// TIA Portal V17 export
// export: Created 2023-08-28T22:41:32.6164324Z, ExportSetting WithDefaults, DisplayName Totally Integrated Automation Portal, DisplayVersion V17 Update 5, DisplayName TIA Portal Openness, DisplayVersion V17 Update 5, DisplayName TIA Portal Teamcenter Gateway, DisplayVersion V17 Update 5, DisplayName TIA Portal Version Control Interface, DisplayVersion V17, DisplayName Simotion SCOUT TIA, DisplayVersion 5.4.3.0, DisplayName TIA Portal Test Suite Advanced, DisplayVersion V17 Update 1, DisplayName SIMOCODE ES, DisplayVersion V17 Update 5, DisplayName SINAMICS Startdrive Advanced, DisplayVersion V17 SP1, DisplayName SINAMICS Startdrive G130, G150, S120, S150, SINAMICS MV, S210, DisplayVersion V17 SP1, DisplayName SINAMICS Startdrive G110M, G120, G120C, G120D, G120P, G115D, DisplayVersion V17 SP1, DisplayName SIRIUS Safety ES, DisplayVersion V17 Update 5, DisplayName STEP 7 Professional, DisplayVersion V17 Update 5, DisplayName STEP 7 CFC, DisplayVersion V17 Update 1, DisplayName STEP 7 Safety, DisplayVersion V17, DisplayName WinCC Advanced, DisplayVersion V17 Update 5, DisplayName SIMATIC Visualization Architect, DisplayVersion V17 Update 5
DATA_BLOCK "S1.CABINET000.STATE"   // DB2700
// stored: AutoNumber true, DBAccessibleFromOPCUA true, DBAccessibleFromWebserver true, InstanceOfName CabState, InstanceOfType FB
"CabState "
BEGIN
END_DATA_BLOCK

DATA_BLOCK "S1.CABINET001.STATE"   // DB2701
// stored: AutoNumber true, DBAccessibleFromOPCUA true, DBAccessibleFromWebserver true, InstanceOfName CabState, InstanceOfType FB
"CabState "
BEGIN
END_DATA_BLOCK

DATA_BLOCK "S1.CABINET002.STATE"   // DB2702
// stored: AutoNumber true, DBAccessibleFromOPCUA true, DBAccessibleFromWebserver true, InstanceOfName CabState, InstanceOfType FB
"CabState "
BEGIN
END_DATA_BLOCK

DATA_BLOCK "S1.CABINET003.STATE"   // DB2703
// stored: AutoNumber true, DBAccessibleFromOPCUA true, DBAccessibleFromWebserver true, InstanceOfName CabState, InstanceOfType FB
"CabState "
BEGIN
END_DATA_BLOCK

DATA_BLOCK "S1.CABINET004.STATE"   // DB2704
// stored: AutoNumber true, DBAccessibleFromOPCUA true, DBAccessibleFromWebserver true, InstanceOfName CabState, InstanceOfType FB
"CabState "
BEGIN
END_DATA_BLOCK

DATA_BLOCK "S1.CABINET005.STATE"   // DB2705
// stored: AutoNumber true, DBAccessibleFromOPCUA true, DBAccessibleFromWebserver true, InstanceOfName CabState, InstanceOfType FB
"CabState "
BEGIN
END_DATA_BLOCK

DATA_BLOCK "S1.CABINET006.STATE"   // DB2706
// stored: AutoNumber true, DBAccessibleFromOPCUA true, DBAccessibleFromWebserver true, InstanceOfName CabState, InstanceOfType FB
"CabState "
BEGIN
END_DATA_BLOCK

DATA_BLOCK "S1.CABINET007.STATE"   // DB2707
// stored: AutoNumber true, DBAccessibleFromOPCUA true, DBAccessibleFromWebserver true, InstanceOfName CabState, InstanceOfType FB
"CabState "
BEGIN
END_DATA_BLOCK

DATA_BLOCK "S1.CABINET008.STATE"   // DB2708
// stored: AutoNumber true, DBAccessibleFromOPCUA true, DBAccessibleFromWebserver true, InstanceOfName CabState, InstanceOfType FB
"CabState "
BEGIN
END_DATA_BLOCK

DATA_BLOCK "S1.CABINET009.STATE"   // DB2709
// stored: AutoNumber true, DBAccessibleFromOPCUA true, DBAccessibleFromWebserver true, InstanceOfName CabState, InstanceOfType FB
"CabState "
BEGIN
END_DATA_BLOCK

DATA_BLOCK "S1.CABINET010.STATE"   // DB2710
// stored: AutoNumber true, DBAccessibleFromOPCUA true, DBAccessibleFromWebserver true, InstanceOfName CabState, InstanceOfType FB
"CabState "
BEGIN
END_DATA_BLOCK

DATA_BLOCK "S1.CABINET011.STATE"   // DB2711
// stored: AutoNumber true, DBAccessibleFromOPCUA true, DBAccessibleFromWebserver true, InstanceOfName CabState, InstanceOfType FB
"CabState "
BEGIN
END_DATA_BLOCK

DATA_BLOCK "S1.CABINET012.STATE"   // DB2712
// stored: AutoNumber true, DBAccessibleFromOPCUA true, DBAccessibleFromWebserver true, InstanceOfName CabState, InstanceOfType FB
"CabState "
BEGIN
END_DATA_BLOCK

DATA_BLOCK "S1.CABINET013.STATE"   // DB2713
// stored: AutoNumber true, DBAccessibleFromOPCUA true, DBAccessibleFromWebserver true, InstanceOfName CabState, InstanceOfType FB
"CabState "
BEGIN
END_DATA_BLOCK

DATA_BLOCK "S1.CABINET014.STATE"   // DB2714
// stored: AutoNumber true, DBAccessibleFromOPCUA true, DBAccessibleFromWebserver true, InstanceOfName CabState, InstanceOfType FB
"CabState "
BEGIN
END_DATA_BLOCK

DATA_BLOCK "S1.CABINET015.STATE"   // DB2715
// stored: AutoNumber true, DBAccessibleFromOPCUA true, DBAccessibleFromWebserver true, InstanceOfName CabState, InstanceOfType FB
"CabState "
BEGIN
END_DATA_BLOCK

DATA_BLOCK "S1.CABINET016.STATE"   // DB2716
// stored: AutoNumber true, DBAccessibleFromOPCUA true, DBAccessibleFromWebserver true, InstanceOfName CabState, InstanceOfType FB
"CabState "
BEGIN
END_DATA_BLOCK

DATA_BLOCK "S1.CABINET017.STATE"   // DB2717
// stored: AutoNumber true, DBAccessibleFromOPCUA true, DBAccessibleFromWebserver true, InstanceOfName CabState, InstanceOfType FB
"CabState "
BEGIN
END_DATA_BLOCK

DATA_BLOCK "S1.CABINET018.STATE"   // DB2718
// stored: AutoNumber true, DBAccessibleFromOPCUA true, DBAccessibleFromWebserver true, InstanceOfName CabState, InstanceOfType FB
"CabState "
BEGIN
END_DATA_BLOCK

DATA_BLOCK "S1.CABINET019.STATE"   // DB2719
// stored: AutoNumber true, DBAccessibleFromOPCUA true, DBAccessibleFromWebserver true, InstanceOfName CabState, InstanceOfType FB
"CabState "
BEGIN
END_DATA_BLOCK

DATA_BLOCK "S1.CABINET020.STATE"   // DB2720
// stored: AutoNumber true, DBAccessibleFromOPCUA true, DBAccessibleFromWebserver true, InstanceOfName CabState, InstanceOfType FB
"CabState "
BEGIN
END_DATA_BLOCK

DATA_BLOCK "S1.CABINET021.STATE"   // DB2721
// stored: AutoNumber true, DBAccessibleFromOPCUA true, DBAccessibleFromWebserver true, InstanceOfName CabState, InstanceOfType FB
"CabState "
BEGIN
END_DATA_BLOCK

DATA_BLOCK "S1.CABINET022.STATE"   // DB2722
// stored: AutoNumber true, DBAccessibleFromOPCUA true, DBAccessibleFromWebserver true, InstanceOfName CabState, InstanceOfType FB
"CabState "
BEGIN
END_DATA_BLOCK

DATA_BLOCK "S1.CABINET023.STATE"   // DB2723
// stored: AutoNumber true, DBAccessibleFromOPCUA true, DBAccessibleFromWebserver true, InstanceOfName CabState, InstanceOfType FB
"CabState "
BEGIN
END_DATA_BLOCK

DATA_BLOCK "S1.CABINET024.STATE"   // DB2724
// stored: AutoNumber true, DBAccessibleFromOPCUA true, DBAccessibleFromWebserver true, InstanceOfName CabState, InstanceOfType FB
"CabState "
BEGIN
END_DATA_BLOCK

DATA_BLOCK "S1.CABINET025.STATE"   // DB2725
// stored: AutoNumber true, DBAccessibleFromOPCUA true, DBAccessibleFromWebserver true, InstanceOfName CabState, InstanceOfType FB
"CabState "
BEGIN
END_DATA_BLOCK

DATA_BLOCK "S1.CABINET026.STATE"   // DB2726
// stored: AutoNumber true, DBAccessibleFromOPCUA true, DBAccessibleFromWebserver true, InstanceOfName CabState, InstanceOfType FB
"CabState "
BEGIN
END_DATA_BLOCK

DATA_BLOCK "S1.CABINET027.STATE"   // DB2727
// stored: AutoNumber true, DBAccessibleFromOPCUA true, DBAccessibleFromWebserver true, InstanceOfName CabState, InstanceOfType FB
"CabState "
BEGIN
END_DATA_BLOCK

DATA_BLOCK "S1.CABINET028.STATE"   // DB2728
// stored: AutoNumber true, DBAccessibleFromOPCUA true, DBAccessibleFromWebserver true, InstanceOfName CabState, InstanceOfType FB
"CabState "
BEGIN
END_DATA_BLOCK

DATA_BLOCK "S1.CABINET029.STATE"   // DB2729
// stored: AutoNumber true, DBAccessibleFromOPCUA true, DBAccessibleFromWebserver true, InstanceOfName CabState, InstanceOfType FB
"CabState "
BEGIN
END_DATA_BLOCK

DATA_BLOCK "S1.CABINET030.STATE"   // DB2730
// stored: AutoNumber true, DBAccessibleFromOPCUA true, DBAccessibleFromWebserver true, InstanceOfName CabState, InstanceOfType FB
"CabState "
BEGIN
END_DATA_BLOCK

DATA_BLOCK "S1.CABINET031.STATE"   // DB2731
// stored: AutoNumber true, DBAccessibleFromOPCUA true, DBAccessibleFromWebserver true, InstanceOfName CabState, InstanceOfType FB
"CabState "
BEGIN
END_DATA_BLOCK

DATA_BLOCK "S1.CABINET032.STATE"   // DB2732
// stored: AutoNumber true, DBAccessibleFromOPCUA true, DBAccessibleFromWebserver true, InstanceOfName CabState, InstanceOfType FB
"CabState "
BEGIN
END_DATA_BLOCK

DATA_BLOCK "S1.CABINET033.STATE"   // DB2733
// stored: AutoNumber true, DBAccessibleFromOPCUA true, DBAccessibleFromWebserver true, InstanceOfName CabState, InstanceOfType FB
"CabState "
BEGIN
END_DATA_BLOCK

DATA_BLOCK "S1.CABINET034.STATE"   // DB2734
// stored: AutoNumber true, DBAccessibleFromOPCUA true, DBAccessibleFromWebserver true, InstanceOfName CabState, InstanceOfType FB
"CabState "
BEGIN
END_DATA_BLOCK

DATA_BLOCK "S1.CABINET035.STATE"   // DB2735
// stored: AutoNumber true, DBAccessibleFromOPCUA true, DBAccessibleFromWebserver true, InstanceOfName CabState, InstanceOfType FB
"CabState "
BEGIN
END_DATA_BLOCK

DATA_BLOCK "S1.CABINET036.STATE"   // DB2736
// stored: AutoNumber true, DBAccessibleFromOPCUA true, DBAccessibleFromWebserver true, InstanceOfName CabState, InstanceOfType FB
"CabState "
BEGIN
END_DATA_BLOCK

DATA_BLOCK "S1.CABINET037.STATE"   // DB2737
// stored: AutoNumber true, DBAccessibleFromOPCUA true, DBAccessibleFromWebserver true, InstanceOfName CabState, InstanceOfType FB
"CabState "
BEGIN
END_DATA_BLOCK

DATA_BLOCK "S1.CABINET038.STATE"   // DB2738
// stored: AutoNumber true, DBAccessibleFromOPCUA true, DBAccessibleFromWebserver true, InstanceOfName CabState, InstanceOfType FB
"CabState "
BEGIN
END_DATA_BLOCK

DATA_BLOCK "S1.CABINET039.STATE"   // DB2739
// stored: AutoNumber true, DBAccessibleFromOPCUA true, DBAccessibleFromWebserver true, InstanceOfName CabState, InstanceOfType FB
"CabState "
BEGIN
END_DATA_BLOCK

DATA_BLOCK "S1.CABINET040.STATE"   // DB2740
// stored: AutoNumber true, DBAccessibleFromOPCUA true, DBAccessibleFromWebserver true, InstanceOfName CabState, InstanceOfType FB
"CabState "
BEGIN
END_DATA_BLOCK

DATA_BLOCK "S1.CABINET041.STATE"   // DB2741
// stored: AutoNumber true, DBAccessibleFromOPCUA true, DBAccessibleFromWebserver true, InstanceOfName CabState, InstanceOfType FB
"CabState "
BEGIN
END_DATA_BLOCK

DATA_BLOCK "S1.CABINET042.STATE"   // DB2742
// stored: AutoNumber true, DBAccessibleFromOPCUA true, DBAccessibleFromWebserver true, InstanceOfName CabState, InstanceOfType FB
"CabState "
BEGIN
END_DATA_BLOCK

DATA_BLOCK "S1.CABINET043.STATE"   // DB2743
// stored: AutoNumber true, DBAccessibleFromOPCUA true, DBAccessibleFromWebserver true, InstanceOfName CabState, InstanceOfType FB
"CabState "
BEGIN
END_DATA_BLOCK

DATA_BLOCK "S1.CABINET044.STATE"   // DB2744
// stored: AutoNumber true, DBAccessibleFromOPCUA true, DBAccessibleFromWebserver true, InstanceOfName CabState, InstanceOfType FB
"CabState "
BEGIN
END_DATA_BLOCK

DATA_BLOCK "S1.CABINET045.STATE"   // DB2745
// stored: AutoNumber true, DBAccessibleFromOPCUA true, DBAccessibleFromWebserver true, InstanceOfName CabState, InstanceOfType FB
"CabState "
BEGIN
END_DATA_BLOCK

DATA_BLOCK "S1.CABINET046.STATE"   // DB2746
// stored: AutoNumber true, DBAccessibleFromOPCUA true, DBAccessibleFromWebserver true, InstanceOfName CabState, InstanceOfType FB
"CabState "
BEGIN
END_DATA_BLOCK

DATA_BLOCK "S1.CABINET047.STATE"   // DB2747
// stored: AutoNumber true, DBAccessibleFromOPCUA true, DBAccessibleFromWebserver true, InstanceOfName CabState, InstanceOfType FB
"CabState "
BEGIN
END_DATA_BLOCK

DATA_BLOCK "S1.CABINET048.STATE"   // DB2748
// stored: AutoNumber true, DBAccessibleFromOPCUA true, DBAccessibleFromWebserver true, InstanceOfName CabState, InstanceOfType FB
"CabState "
BEGIN
END_DATA_BLOCK

DATA_BLOCK "S1.CABINET049.STATE"   // DB2749
// stored: AutoNumber true, DBAccessibleFromOPCUA true, DBAccessibleFromWebserver true, InstanceOfName CabState, InstanceOfType FB
"CabState "
BEGIN
END_DATA_BLOCK

DATA_BLOCK "S1.CABINET050.STATE"   // DB2750
// stored: AutoNumber true, DBAccessibleFromOPCUA true, DBAccessibleFromWebserver true, InstanceOfName CabState, InstanceOfType FB
"CabState "
BEGIN
END_DATA_BLOCK

DATA_BLOCK "S1.CABINET051.STATE"   // DB2751
// stored: AutoNumber true, DBAccessibleFromOPCUA true, DBAccessibleFromWebserver true, InstanceOfName CabState, InstanceOfType FB
"CabState "
BEGIN
END_DATA_BLOCK

DATA_BLOCK "S1.CABINET052.STATE"   // DB2752
// stored: AutoNumber true, DBAccessibleFromOPCUA true, DBAccessibleFromWebserver true, InstanceOfName CabState, InstanceOfType FB
"CabState "
BEGIN
END_DATA_BLOCK

DATA_BLOCK "S1.CABINET053.STATE"   // DB2753
// stored: AutoNumber true, DBAccessibleFromOPCUA true, DBAccessibleFromWebserver true, InstanceOfName CabState, InstanceOfType FB
"CabState "
BEGIN
END_DATA_BLOCK

DATA_BLOCK "S1.CABINET054.STATE"   // DB2754
// stored: AutoNumber true, DBAccessibleFromOPCUA true, DBAccessibleFromWebserver true, InstanceOfName CabState, InstanceOfType FB
"CabState "
BEGIN
END_DATA_BLOCK

DATA_BLOCK "S1.CABINET055.STATE"   // DB2755
// stored: AutoNumber true, DBAccessibleFromOPCUA true, DBAccessibleFromWebserver true, InstanceOfName CabState, InstanceOfType FB
"CabState "
BEGIN
END_DATA_BLOCK

DATA_BLOCK "S1.CABINET056.STATE"   // DB2756
// stored: AutoNumber true, DBAccessibleFromOPCUA true, DBAccessibleFromWebserver true, InstanceOfName CabState, InstanceOfType FB
"CabState "
BEGIN
END_DATA_BLOCK

DATA_BLOCK "S1.CABINET057.STATE"   // DB2757
// stored: AutoNumber true, DBAccessibleFromOPCUA true, DBAccessibleFromWebserver true, InstanceOfName CabState, InstanceOfType FB
"CabState "
BEGIN
END_DATA_BLOCK

DATA_BLOCK "S1.CABINET058.STATE"   // DB2758
// stored: AutoNumber true, DBAccessibleFromOPCUA true, DBAccessibleFromWebserver true, InstanceOfName CabState, InstanceOfType FB
"CabState "
BEGIN
END_DATA_BLOCK

DATA_BLOCK "S1.CABINET059.STATE"   // DB2759
// stored: AutoNumber true, DBAccessibleFromOPCUA true, DBAccessibleFromWebserver true, InstanceOfName CabState, InstanceOfType FB
"CabState "
BEGIN
END_DATA_BLOCK

DATA_BLOCK "S1.CABINET060.STATE"   // DB2760
// stored: AutoNumber true, DBAccessibleFromOPCUA true, DBAccessibleFromWebserver true, InstanceOfName CabState, InstanceOfType FB
"CabState "
BEGIN
END_DATA_BLOCK

DATA_BLOCK "S1.CABINET061.STATE"   // DB2761
// stored: AutoNumber true, DBAccessibleFromOPCUA true, DBAccessibleFromWebserver true, InstanceOfName CabState, InstanceOfType FB
"CabState "
BEGIN
END_DATA_BLOCK

DATA_BLOCK "S1.CABINET062.STATE"   // DB2762
// stored: AutoNumber true, DBAccessibleFromOPCUA true, DBAccessibleFromWebserver true, InstanceOfName CabState, InstanceOfType FB
"CabState "
BEGIN
END_DATA_BLOCK

DATA_BLOCK "S1.CABINET063.STATE"   // DB2763
// stored: AutoNumber true, DBAccessibleFromOPCUA true, DBAccessibleFromWebserver true, InstanceOfName CabState, InstanceOfType FB
"CabState "
BEGIN
END_DATA_BLOCK

DATA_BLOCK "S1.CABINET064.STATE"   // DB2764
// stored: AutoNumber true, DBAccessibleFromOPCUA true, DBAccessibleFromWebserver true, InstanceOfName CabState, InstanceOfType FB
"CabState "
BEGIN
END_DATA_BLOCK

DATA_BLOCK "S1.CABINET065.STATE"   // DB2765
// stored: AutoNumber true, DBAccessibleFromOPCUA true, DBAccessibleFromWebserver true, InstanceOfName CabState, InstanceOfType FB
"CabState "
BEGIN
END_DATA_BLOCK

DATA_BLOCK "S1.CABINET066.STATE"   // DB2766
// stored: AutoNumber true, DBAccessibleFromOPCUA true, DBAccessibleFromWebserver true, InstanceOfName CabState, InstanceOfType FB
"CabState "
BEGIN
END_DATA_BLOCK

DATA_BLOCK "S1.CABINET067.STATE"   // DB2767
// stored: AutoNumber true, DBAccessibleFromOPCUA true, DBAccessibleFromWebserver true, InstanceOfName CabState, InstanceOfType FB
"CabState "
BEGIN
END_DATA_BLOCK

DATA_BLOCK "S1.CABINET068.STATE"   // DB2768
// stored: AutoNumber true, DBAccessibleFromOPCUA true, DBAccessibleFromWebserver true, InstanceOfName CabState, InstanceOfType FB
"CabState "
BEGIN
END_DATA_BLOCK

DATA_BLOCK "S1.CABINET069.STATE"   // DB2769
// stored: AutoNumber true, DBAccessibleFromOPCUA true, DBAccessibleFromWebserver true, InstanceOfName CabState, InstanceOfType FB
"CabState "
BEGIN
END_DATA_BLOCK

DATA_BLOCK "S1.CABINET070.STATE"   // DB2770
// stored: AutoNumber true, DBAccessibleFromOPCUA true, DBAccessibleFromWebserver true, InstanceOfName CabState, InstanceOfType FB
"CabState "
BEGIN
END_DATA_BLOCK

DATA_BLOCK "S1.CABINET071.STATE"   // DB2771
// stored: AutoNumber true, DBAccessibleFromOPCUA true, DBAccessibleFromWebserver true, InstanceOfName CabState, InstanceOfType FB
"CabState "
BEGIN
END_DATA_BLOCK

DATA_BLOCK "S1.CABINET072.STATE"   // DB2772
// stored: AutoNumber true, DBAccessibleFromOPCUA true, DBAccessibleFromWebserver true, InstanceOfName CabState, InstanceOfType FB
"CabState "
BEGIN
END_DATA_BLOCK

DATA_BLOCK "S1.CABINET073.STATE"   // DB2773
// stored: AutoNumber true, DBAccessibleFromOPCUA true, DBAccessibleFromWebserver true, InstanceOfName CabState, InstanceOfType FB
"CabState "
BEGIN
END_DATA_BLOCK

DATA_BLOCK "S1.CABINET074.STATE"   // DB2774
// stored: AutoNumber true, DBAccessibleFromOPCUA true, DBAccessibleFromWebserver true, InstanceOfName CabState, InstanceOfType FB
"CabState "
BEGIN
END_DATA_BLOCK

DATA_BLOCK "S1.CABINET075.STATE"   // DB2775
// stored: AutoNumber true, DBAccessibleFromOPCUA true, DBAccessibleFromWebserver true, InstanceOfName CabState, InstanceOfType FB
"CabState "
BEGIN
END_DATA_BLOCK

DATA_BLOCK "S1.CABINET076.STATE"   // DB2776
// stored: AutoNumber true, DBAccessibleFromOPCUA true, DBAccessibleFromWebserver true, InstanceOfName CabState, InstanceOfType FB
"CabState "
BEGIN
END_DATA_BLOCK

DATA_BLOCK "S1.CABINET077.STATE"   // DB2777
// stored: AutoNumber true, DBAccessibleFromOPCUA true, DBAccessibleFromWebserver true, InstanceOfName CabState, InstanceOfType FB
"CabState "
BEGIN
END_DATA_BLOCK

DATA_BLOCK "S1.CABINET078.STATE"   // DB2778
// stored: AutoNumber true, DBAccessibleFromOPCUA true, DBAccessibleFromWebserver true, InstanceOfName CabState, InstanceOfType FB
"CabState "
BEGIN
END_DATA_BLOCK

DATA_BLOCK "S1.CABINET079.STATE"   // DB2779
// stored: AutoNumber true, DBAccessibleFromOPCUA true, DBAccessibleFromWebserver true, InstanceOfName CabState, InstanceOfType FB
"CabState "
BEGIN
END_DATA_BLOCK

DATA_BLOCK "S1.CABINET080.STATE"   // DB2780
// stored: AutoNumber true, DBAccessibleFromOPCUA true, DBAccessibleFromWebserver true, InstanceOfName CabState, InstanceOfType FB
"CabState "
BEGIN
END_DATA_BLOCK

DATA_BLOCK "S1.CABINET081.STATE"   // DB2781
// stored: AutoNumber true, DBAccessibleFromOPCUA true, DBAccessibleFromWebserver true, InstanceOfName CabState, InstanceOfType FB
"CabState "
BEGIN
END_DATA_BLOCK

DATA_BLOCK "S1.CABINET082.STATE"   // DB2782
// stored: AutoNumber true, DBAccessibleFromOPCUA true, DBAccessibleFromWebserver true, InstanceOfName CabState, InstanceOfType FB
"CabState "
BEGIN
END_DATA_BLOCK

DATA_BLOCK "S1.CABINET083.STATE"   // DB2783
// stored: AutoNumber true, DBAccessibleFromOPCUA true, DBAccessibleFromWebserver true, InstanceOfName CabState, InstanceOfType FB
"CabState "
BEGIN
END_DATA_BLOCK

DATA_BLOCK "S1.CABINET084.STATE"   // DB2784
// stored: AutoNumber true, DBAccessibleFromOPCUA true, DBAccessibleFromWebserver true, InstanceOfName CabState, InstanceOfType FB
"CabState "
BEGIN
END_DATA_BLOCK

DATA_BLOCK "S1.CABINET085.STATE"   // DB2785
// stored: AutoNumber true, DBAccessibleFromOPCUA true, DBAccessibleFromWebserver true, InstanceOfName CabState, InstanceOfType FB
"CabState "
BEGIN
END_DATA_BLOCK

DATA_BLOCK "S1.CABINET086.STATE"   // DB2786
// stored: AutoNumber true, DBAccessibleFromOPCUA true, DBAccessibleFromWebserver true, InstanceOfName CabState, InstanceOfType FB
"CabState "
BEGIN
END_DATA_BLOCK

DATA_BLOCK "S1.CABINET087.STATE"   // DB2787
// stored: AutoNumber true, DBAccessibleFromOPCUA true, DBAccessibleFromWebserver true, InstanceOfName CabState, InstanceOfType FB
"CabState "
BEGIN
END_DATA_BLOCK

DATA_BLOCK "S1.CABINET088.STATE"   // DB2788
// stored: AutoNumber true, DBAccessibleFromOPCUA true, DBAccessibleFromWebserver true, InstanceOfName CabState, InstanceOfType FB
"CabState "
BEGIN
END_DATA_BLOCK

DATA_BLOCK "S1.CABINET089.STATE"   // DB2789
// stored: AutoNumber true, DBAccessibleFromOPCUA true, DBAccessibleFromWebserver true, InstanceOfName CabState, InstanceOfType FB
"CabState "
BEGIN
END_DATA_BLOCK

DATA_BLOCK "S1.CABINET090.STATE"   // DB2790
// stored: AutoNumber true, DBAccessibleFromOPCUA true, DBAccessibleFromWebserver true, InstanceOfName CabState, InstanceOfType FB
"CabState "
BEGIN
END_DATA_BLOCK

DATA_BLOCK "S1.CABINET091.STATE"   // DB2791
// stored: AutoNumber true, DBAccessibleFromOPCUA true, DBAccessibleFromWebserver true, InstanceOfName CabState, InstanceOfType FB
"CabState "
BEGIN
END_DATA_BLOCK

DATA_BLOCK "S1.CABINET092.STATE"   // DB2792
// stored: AutoNumber true, DBAccessibleFromOPCUA true, DBAccessibleFromWebserver true, InstanceOfName CabState, InstanceOfType FB
"CabState "
BEGIN
END_DATA_BLOCK

DATA_BLOCK "S1.CABINET093.STATE"   // DB2793
// stored: AutoNumber true, DBAccessibleFromOPCUA true, DBAccessibleFromWebserver true, InstanceOfName CabState, InstanceOfType FB
"CabState "
BEGIN
END_DATA_BLOCK

DATA_BLOCK "S1.CABINET094.STATE"   // DB2794
// stored: AutoNumber true, DBAccessibleFromOPCUA true, DBAccessibleFromWebserver true, InstanceOfName CabState, InstanceOfType FB
"CabState "
BEGIN
END_DATA_BLOCK

DATA_BLOCK "S1.CABINET095.STATE"   // DB2795
// stored: AutoNumber true, DBAccessibleFromOPCUA true, DBAccessibleFromWebserver true, InstanceOfName CabState, InstanceOfType FB
"CabState "
BEGIN
END_DATA_BLOCK

DATA_BLOCK "S1.CABINET096.STATE"   // DB2796
// stored: AutoNumber true, DBAccessibleFromOPCUA true, DBAccessibleFromWebserver true, InstanceOfName CabState, InstanceOfType FB
"CabState "
BEGIN
END_DATA_BLOCK

DATA_BLOCK "S1.CABINET097.STATE"   // DB2797
// stored: AutoNumber true, DBAccessibleFromOPCUA true, DBAccessibleFromWebserver true, InstanceOfName CabState, InstanceOfType FB
"CabState "
BEGIN
END_DATA_BLOCK

DATA_BLOCK "S1.CABINET098.STATE"   // DB2798
// stored: AutoNumber true, DBAccessibleFromOPCUA true, DBAccessibleFromWebserver true, InstanceOfName CabState, InstanceOfType FB
"CabState "
BEGIN
END_DATA_BLOCK

DATA_BLOCK "S1.CABINET099.STATE"   // DB2799
// stored: AutoNumber true, DBAccessibleFromOPCUA true, DBAccessibleFromWebserver true, InstanceOfName CabState, InstanceOfType FB
"CabState "
BEGIN
END_DATA_BLOCK

DATA_BLOCK "S1.CABINET100.STATE"   // DB2800
// stored: AutoNumber true, DBAccessibleFromOPCUA true, DBAccessibleFromWebserver true, InstanceOfName CabState, InstanceOfType FB
"CabState "
BEGIN
END_DATA_BLOCK

DATA_BLOCK "S1.CABINET101.STATE"   // DB2801
// stored: AutoNumber true, DBAccessibleFromOPCUA true, DBAccessibleFromWebserver true, InstanceOfName CabState, InstanceOfType FB
"CabState "
BEGIN
END_DATA_BLOCK

DATA_BLOCK "S1.CABINET102.STATE"   // DB2802
// stored: AutoNumber true, DBAccessibleFromOPCUA true, DBAccessibleFromWebserver true, InstanceOfName CabState, InstanceOfType FB
"CabState "
BEGIN
END_DATA_BLOCK

DATA_BLOCK "S1.CABINET103.STATE"   // DB2803
// stored: AutoNumber true, DBAccessibleFromOPCUA true, DBAccessibleFromWebserver true, InstanceOfName CabState, InstanceOfType FB
"CabState "
BEGIN
END_DATA_BLOCK

DATA_BLOCK "S1.CABINET104.STATE"   // DB2804
// stored: AutoNumber true, DBAccessibleFromOPCUA true, DBAccessibleFromWebserver true, InstanceOfName CabState, InstanceOfType FB
"CabState "
BEGIN
END_DATA_BLOCK

DATA_BLOCK "S1.CABINET105.STATE"   // DB2805
// stored: AutoNumber true, DBAccessibleFromOPCUA true, DBAccessibleFromWebserver true, InstanceOfName CabState, InstanceOfType FB
"CabState "
BEGIN
END_DATA_BLOCK

DATA_BLOCK "S1.CABINET106.STATE"   // DB2806
// stored: AutoNumber true, DBAccessibleFromOPCUA true, DBAccessibleFromWebserver true, InstanceOfName CabState, InstanceOfType FB
"CabState "
BEGIN
END_DATA_BLOCK

DATA_BLOCK "S1.CABINET107.STATE"   // DB2807
// stored: AutoNumber true, DBAccessibleFromOPCUA true, DBAccessibleFromWebserver true, InstanceOfName CabState, InstanceOfType FB
"CabState "
BEGIN
END_DATA_BLOCK

DATA_BLOCK "S1.CABINET108.STATE"   // DB2808
// stored: AutoNumber true, DBAccessibleFromOPCUA true, DBAccessibleFromWebserver true, InstanceOfName CabState, InstanceOfType FB
"CabState "
BEGIN
END_DATA_BLOCK

DATA_BLOCK "S1.CABINET109.STATE"   // DB2809
// stored: AutoNumber true, DBAccessibleFromOPCUA true, DBAccessibleFromWebserver true, InstanceOfName CabState, InstanceOfType FB
"CabState "
BEGIN
END_DATA_BLOCK

DATA_BLOCK "S1.CABINET110.STATE"   // DB2810
// stored: AutoNumber true, DBAccessibleFromOPCUA true, DBAccessibleFromWebserver true, InstanceOfName CabState, InstanceOfType FB
"CabState "
BEGIN
END_DATA_BLOCK

DATA_BLOCK "S1.CABINET111.STATE"   // DB2811
// stored: AutoNumber true, DBAccessibleFromOPCUA true, DBAccessibleFromWebserver true, InstanceOfName CabState, InstanceOfType FB
"CabState "
BEGIN
END_DATA_BLOCK
